{attribute 'qualified_only'}
{attribute 'strict'}
TYPE eNetContactorDirection :
(
	Left 	:= -1,
	None 	:= 0,
	Right 	:= 1
);
END_TYPE

(* stored: Version 1.1.0.1, ProductVersion 3.1.4026.18
   DUT eNetContactorDirection: Id {679310d3-e692-4a42-a743-46b64572b479} *)
